TYPE eTorqueMode :
	(		
		mcFF :=0 ,
		mcLimit 
		
	);
END_TYPE

(* stored: Version 1.1.0.1, ProductVersion 3.1.4024.3
   DUT eTorqueMode: Id {15cb4b3d-132b-4a8d-87df-1e7f84838f37} *)
